PROGRAM P02_GlobalSystemTime
VAR
	fbGlobalTime 		:FB_SystemDateTIme;
	
END_VAR

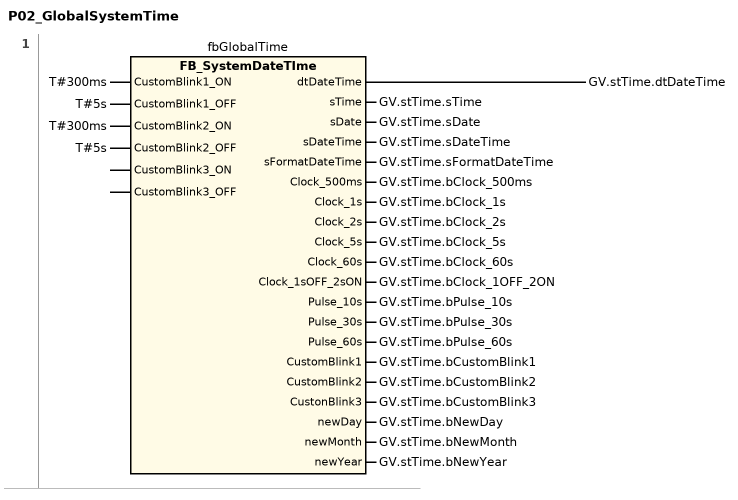
// NETWORK 1
fbGlobalTime(
    CustomBlink1_ON := T#300ms,
    CustomBlink1_OFF := T#5s,
    CustomBlink2_ON := T#300ms,
    CustomBlink2_OFF := T#5s,
    sTime => GV.stTime.sTime,
    sDate => GV.stTime.sDate,
    sDateTime => GV.stTime.sDateTime,
    sFormatDateTime => GV.stTime.sFormatDateTime,
    Clock_500ms => GV.stTime.bClock_500ms,
    Clock_1s => GV.stTime.bClock_1s,
    Clock_2s => GV.stTime.bClock_2s,
    Clock_5s => GV.stTime.bClock_5s,
    Clock_60s => GV.stTime.bClock_60s,
    Clock_1sOFF_2sON => GV.stTime.bClock_1OFF_2ON,
    Pulse_10s => GV.stTime.bPulse_10s,
    Pulse_30s => GV.stTime.bPulse_30s,
    Pulse_60s => GV.stTime.bPulse_60s,
    CustomBlink1 => GV.stTime.bCustomBlink1,
    CustomBlink2 => GV.stTime.bCustomBlink2,
    CustonBlink3 => GV.stTime.bCustomBlink3,
    newDay => GV.stTime.bNewDay,
    newMonth => GV.stTime.bNewMonth,
    newYear => GV.stTime.bNewYear); // FB_SystemDateTIme
GV.stTime.dtDateTime := fbGlobalTime.dtDateTime;

END_PROGRAM

(* stored: Version 1.1.0.1, ProductVersion 3.1.4026.13
   POU P02_GlobalSystemTime: Id {b84d2a5b-18ea-4b9a-ba47-60f0d98102d0}, SpecialFunc None *)
